TYPE ST_SequenceIn :
STRUCT
END_STRUCT
END_TYPE

(* stored: Version 1.1.0.1
   DUT ST_SequenceIn: Id {8bb40e74-574f-0055-2dd6-6a94905152be} *)
